# EPICS autosave request: iocBoot/iocARAmp/auto_settings_ARAmp.req
file "aramp_settings.req",                P=$(P),  R=$(R)
